//!<param name="nNumberOfOutputArguments">determined amount of output parameters</param>

//!<param name="nReserved">Reserved padding</param>

{attribute 'pack_mode' := '1'}
TYPE OPC_UA_OUTPUT_ARGUMENT_INFO_AND_DATA :
STRUCT
	nNumberOfOutputArguments: UDINT; 
	nReserved: ARRAY[1..4] OF BYTE; 
	//stOutputArgInfo: ARRAY[*] OF ST_UAMethodArgInfo; 
	//data : DINT;
END_STRUCT
END_TYPE

(* stored: Version 1.1.0.1
   DUT OPC_UA_OUTPUT_ARGUMENT_INFO_AND_DATA: Id {aa411b33-0ffd-48f8-ad37-0dd63243bc1d} *)
